// TIA Portal V15.1 export
// export: Created 2024-05-17T05:38:55.7336382Z, ExportSetting WithDefaults, DisplayName Totally Integrated Automation Portal, DisplayVersion V15.1 Update 5, DisplayName TIA Portal Openness, DisplayVersion V15.1 Update 5, DisplayName SINAMICS Startdrive Advanced, DisplayVersion V15.1, DisplayName G130, G150, S120, S150, SINAMICS MV, S210, DisplayVersion V15.1, DisplayName G110M, G120, G120C, G120D, G120P, DisplayVersion V15.1, DisplayName STEP 7 Professional, DisplayVersion V15.1 Update 5, DisplayName STEP 7 Safety, DisplayVersion V15.1, DisplayName WinCC Professional, DisplayVersion V15.1 Update 5, DisplayName SIMATIC Visualization Architect, DisplayVersion V15.1
FUNCTION "209220ZM01Andon" : Void   // FC356, FBD
TITLE = 209220ZM01 Andon
{ S7_Optimized_Access := 'FALSE' }
AUTHOR : VCG
NAME : Mot001
VERSION : 0.1
// stored: AutoNumber false, IsIECCheckEnabled false, SetENOAutomatically False, UDAEnableTagReadback false
   VAR_OUTPUT
      O_AlarmA : Bool;   // Alarm A
      O_AlarmB : Bool;   // Alarm B
      O_AlarmC : Bool;   // Alarm C
      O_AlarmD : Bool;   // Alarm D
      O_AlarmABCondition : Bool;   // Alarms resetable
      H_IAnim : Word;   // Animation bits to Icon in WinCC
   END_VAR
BEGIN

REGION Network 1: **** 1 - Inputs **** HMI Commands
   // HMI Commands from the WinCC
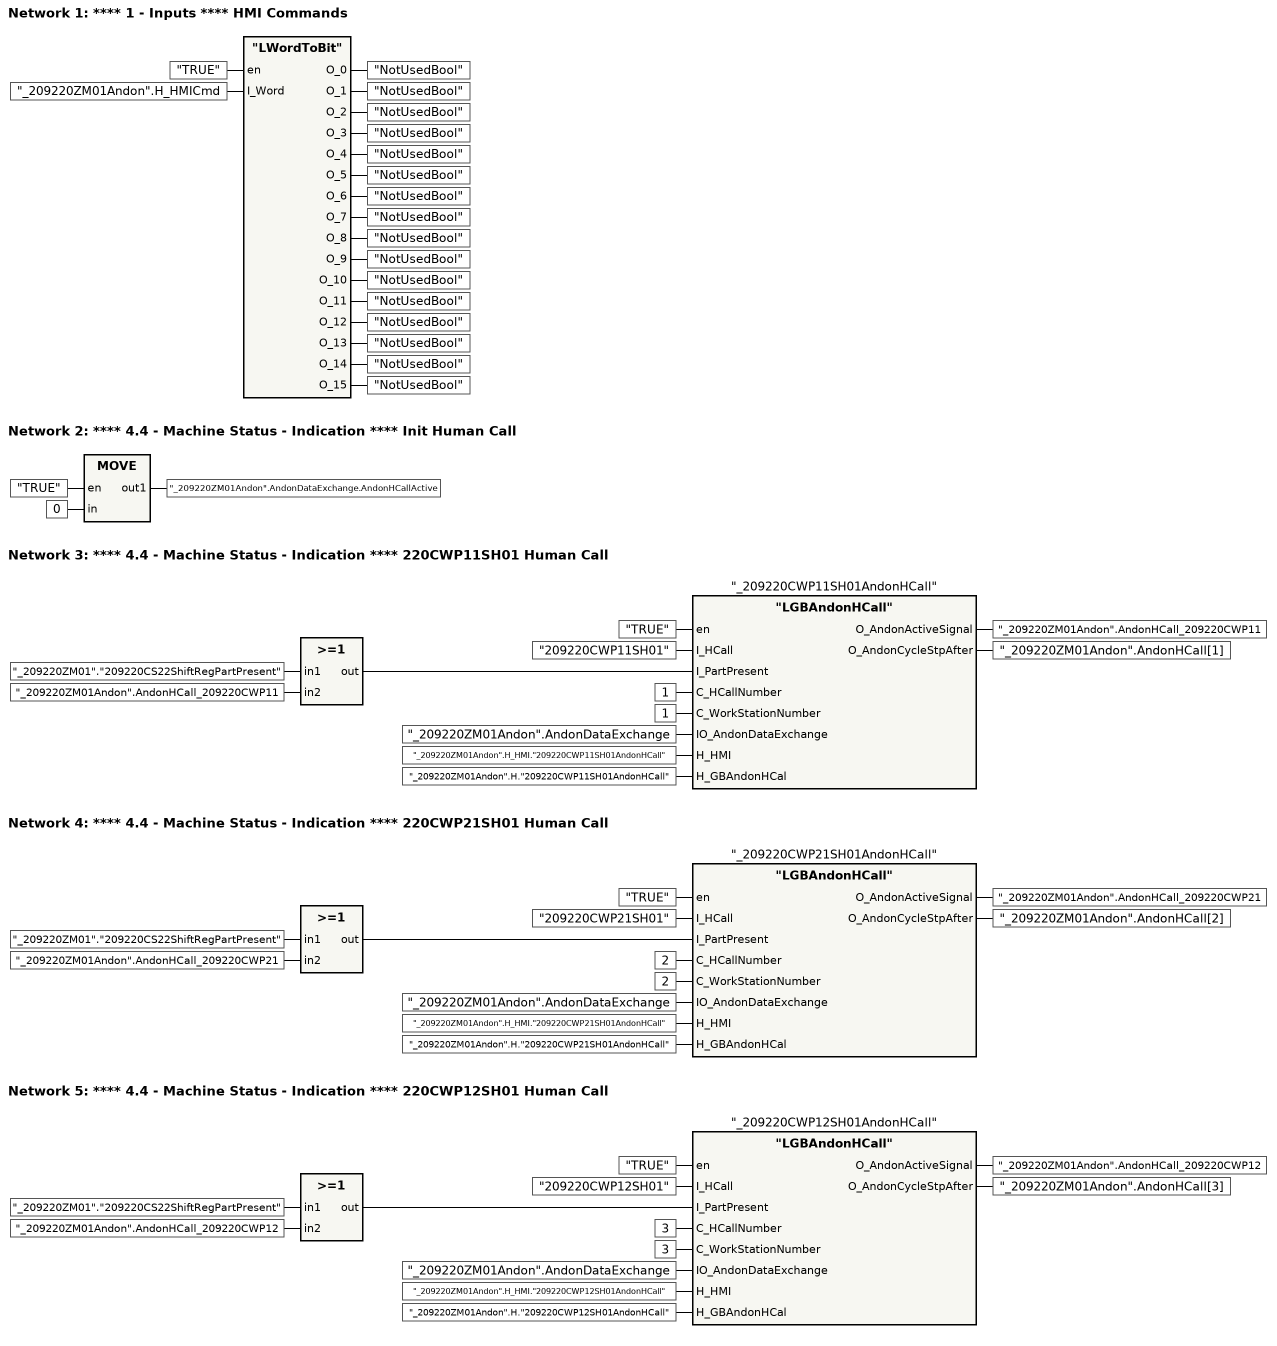
   IF "TRUE" THEN
       "LWordToBit"(I_Word := "_209220ZM01Andon".H_HMICmd,
                    O_0 => "NotUsedBool",
                    O_1 => "NotUsedBool",
                    O_2 => "NotUsedBool",
                    O_3 => "NotUsedBool",
                    O_4 => "NotUsedBool",
                    O_5 => "NotUsedBool",
                    O_6 => "NotUsedBool",
                    O_7 => "NotUsedBool",
                    O_8 => "NotUsedBool",
                    O_9 => "NotUsedBool",
                    O_10 => "NotUsedBool",
                    O_11 => "NotUsedBool",
                    O_12 => "NotUsedBool",
                    O_13 => "NotUsedBool",
                    O_14 => "NotUsedBool",
                    O_15 => "NotUsedBool");
   END_IF;
END_REGION

REGION Network 2: **** 4.4 - Machine Status - Indication **** Init Human Call
   IF "TRUE" THEN "_209220ZM01Andon".AndonDataExchange.AndonHCallActive := 0; END_IF;
END_REGION

REGION Network 3: **** 4.4 - Machine Status - Indication **** 220CWP11SH01 Human Call
   IF "TRUE" THEN
       "_209220CWP11SH01AndonHCall"(I_HCall := "209220CWP11SH01",   // "LGBAndonHCall"
                               I_PartPresent := "_209220ZM01"."209220CS22ShiftRegPartPresent" OR "_209220ZM01Andon".AndonHCall_209220CWP11,
                               C_HCallNumber := 1,
                               C_WorkStationNumber := 1,
                               IO_AndonDataExchange := "_209220ZM01Andon".AndonDataExchange,
                               H_HMI := "_209220ZM01Andon".H_HMI."209220CWP11SH01AndonHCall",
                               H_GBAndonHCal := "_209220ZM01Andon".H."209220CWP11SH01AndonHCall",
                               O_AndonActiveSignal => "_209220ZM01Andon".AndonHCall_209220CWP11,
                               O_AndonCycleStpAfter => "_209220ZM01Andon".AndonHCall[1]);
   END_IF;
END_REGION

REGION Network 4: **** 4.4 - Machine Status - Indication **** 220CWP21SH01 Human Call
   IF "TRUE" THEN
       "_209220CWP21SH01AndonHCall"(I_HCall := "209220CWP21SH01",   // "LGBAndonHCall"
                               I_PartPresent := "_209220ZM01"."209220CS22ShiftRegPartPresent" OR "_209220ZM01Andon".AndonHCall_209220CWP21,
                               C_HCallNumber := 2,
                               C_WorkStationNumber := 2,
                               IO_AndonDataExchange := "_209220ZM01Andon".AndonDataExchange,
                               H_HMI := "_209220ZM01Andon".H_HMI."209220CWP21SH01AndonHCall",
                               H_GBAndonHCal := "_209220ZM01Andon".H."209220CWP21SH01AndonHCall",
                               O_AndonActiveSignal => "_209220ZM01Andon".AndonHCall_209220CWP21,
                               O_AndonCycleStpAfter => "_209220ZM01Andon".AndonHCall[2]);
   END_IF;
END_REGION

REGION Network 5: **** 4.4 - Machine Status - Indication **** 220CWP12SH01 Human Call
   IF "TRUE" THEN
       "_209220CWP12SH01AndonHCall"(I_HCall := "209220CWP12SH01",   // "LGBAndonHCall"
                               I_PartPresent := "_209220ZM01"."209220CS22ShiftRegPartPresent" OR "_209220ZM01Andon".AndonHCall_209220CWP12,
                               C_HCallNumber := 3,
                               C_WorkStationNumber := 3,
                               IO_AndonDataExchange := "_209220ZM01Andon".AndonDataExchange,
                               H_HMI := "_209220ZM01Andon".H_HMI."209220CWP12SH01AndonHCall",
                               H_GBAndonHCal := "_209220ZM01Andon".H."209220CWP12SH01AndonHCall",
                               O_AndonActiveSignal => "_209220ZM01Andon".AndonHCall_209220CWP12,
                               O_AndonCycleStpAfter => "_209220ZM01Andon".AndonHCall[3]);
   END_IF;
END_REGION

REGION Network 6: **** 4.4 - Machine Status - Indication **** 220CWP22SH01 Human Call
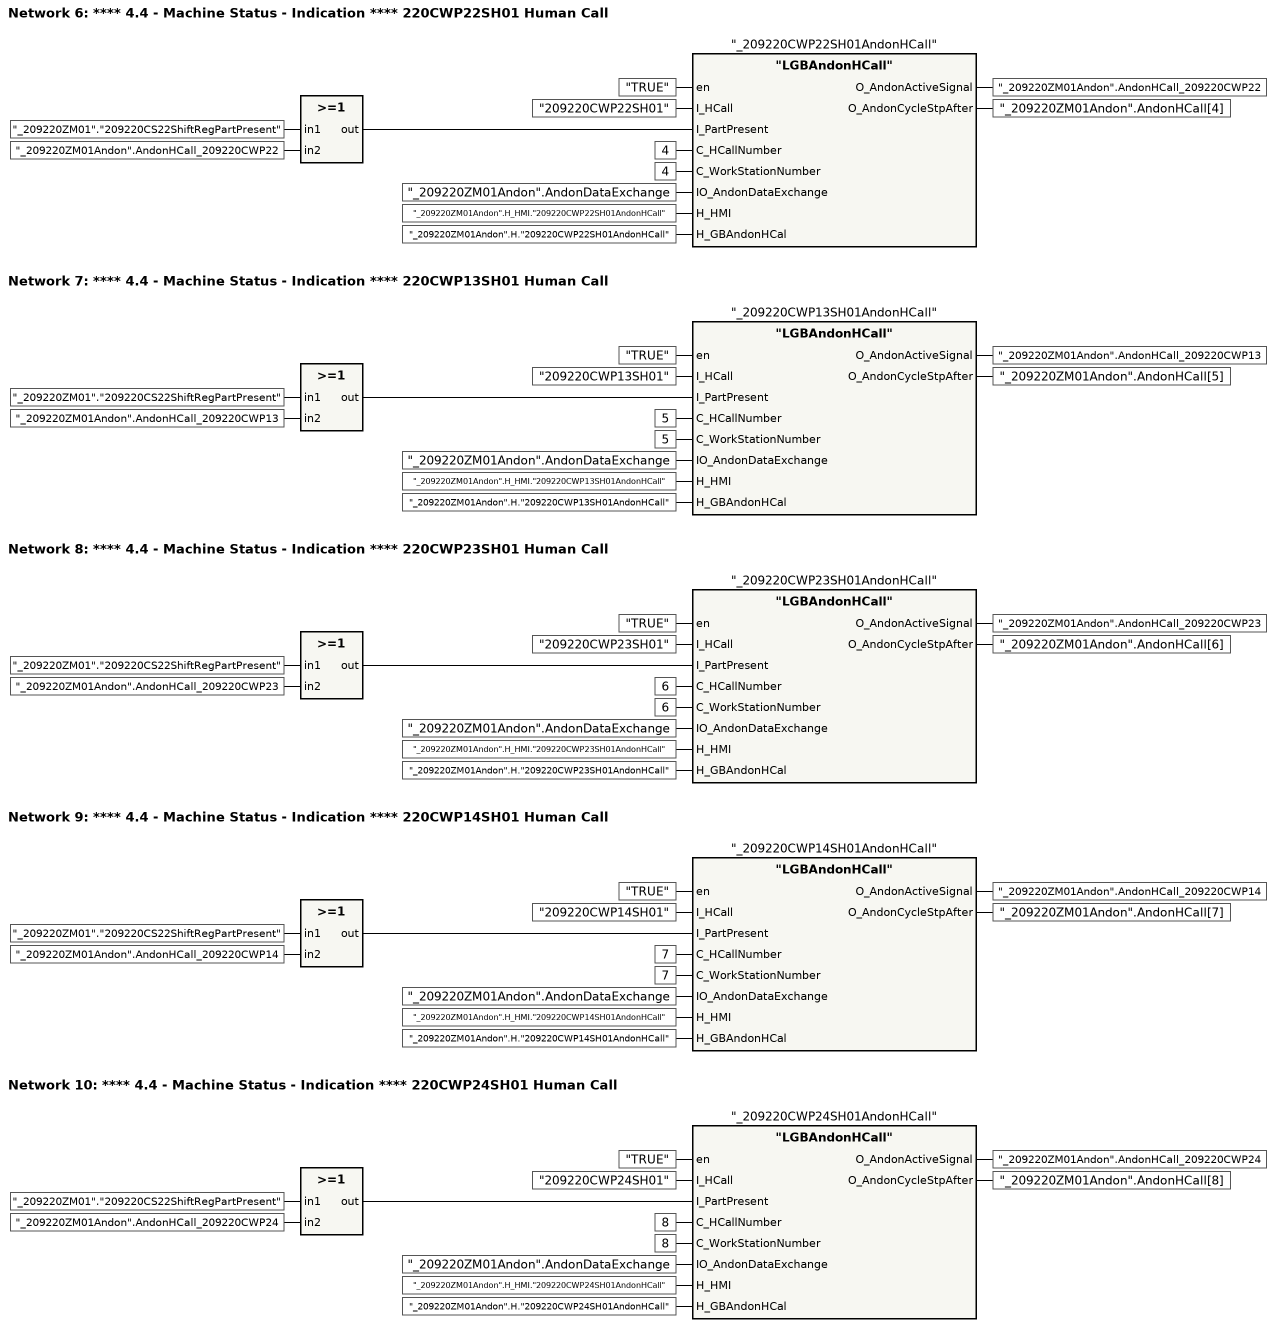
   IF "TRUE" THEN
       "_209220CWP22SH01AndonHCall"(I_HCall := "209220CWP22SH01",   // "LGBAndonHCall"
                               I_PartPresent := "_209220ZM01"."209220CS22ShiftRegPartPresent" OR "_209220ZM01Andon".AndonHCall_209220CWP22,
                               C_HCallNumber := 4,
                               C_WorkStationNumber := 4,
                               IO_AndonDataExchange := "_209220ZM01Andon".AndonDataExchange,
                               H_HMI := "_209220ZM01Andon".H_HMI."209220CWP22SH01AndonHCall",
                               H_GBAndonHCal := "_209220ZM01Andon".H."209220CWP22SH01AndonHCall",
                               O_AndonActiveSignal => "_209220ZM01Andon".AndonHCall_209220CWP22,
                               O_AndonCycleStpAfter => "_209220ZM01Andon".AndonHCall[4]);
   END_IF;
END_REGION

REGION Network 7: **** 4.4 - Machine Status - Indication **** 220CWP13SH01 Human Call
   IF "TRUE" THEN
       "_209220CWP13SH01AndonHCall"(I_HCall := "209220CWP13SH01",   // "LGBAndonHCall"
                               I_PartPresent := "_209220ZM01"."209220CS22ShiftRegPartPresent" OR "_209220ZM01Andon".AndonHCall_209220CWP13,
                               C_HCallNumber := 5,
                               C_WorkStationNumber := 5,
                               IO_AndonDataExchange := "_209220ZM01Andon".AndonDataExchange,
                               H_HMI := "_209220ZM01Andon".H_HMI."209220CWP13SH01AndonHCall",
                               H_GBAndonHCal := "_209220ZM01Andon".H."209220CWP13SH01AndonHCall",
                               O_AndonActiveSignal => "_209220ZM01Andon".AndonHCall_209220CWP13,
                               O_AndonCycleStpAfter => "_209220ZM01Andon".AndonHCall[5]);
   END_IF;
END_REGION

REGION Network 8: **** 4.4 - Machine Status - Indication **** 220CWP23SH01 Human Call
   IF "TRUE" THEN
       "_209220CWP23SH01AndonHCall"(I_HCall := "209220CWP23SH01",   // "LGBAndonHCall"
                               I_PartPresent := "_209220ZM01"."209220CS22ShiftRegPartPresent" OR "_209220ZM01Andon".AndonHCall_209220CWP23,
                               C_HCallNumber := 6,
                               C_WorkStationNumber := 6,
                               IO_AndonDataExchange := "_209220ZM01Andon".AndonDataExchange,
                               H_HMI := "_209220ZM01Andon".H_HMI."209220CWP23SH01AndonHCall",
                               H_GBAndonHCal := "_209220ZM01Andon".H."209220CWP23SH01AndonHCall",
                               O_AndonActiveSignal => "_209220ZM01Andon".AndonHCall_209220CWP23,
                               O_AndonCycleStpAfter => "_209220ZM01Andon".AndonHCall[6]);
   END_IF;
END_REGION

REGION Network 9: **** 4.4 - Machine Status - Indication **** 220CWP14SH01 Human Call
   IF "TRUE" THEN
       "_209220CWP14SH01AndonHCall"(I_HCall := "209220CWP14SH01",   // "LGBAndonHCall"
                               I_PartPresent := "_209220ZM01"."209220CS22ShiftRegPartPresent" OR "_209220ZM01Andon".AndonHCall_209220CWP14,
                               C_HCallNumber := 7,
                               C_WorkStationNumber := 7,
                               IO_AndonDataExchange := "_209220ZM01Andon".AndonDataExchange,
                               H_HMI := "_209220ZM01Andon".H_HMI."209220CWP14SH01AndonHCall",
                               H_GBAndonHCal := "_209220ZM01Andon".H."209220CWP14SH01AndonHCall",
                               O_AndonActiveSignal => "_209220ZM01Andon".AndonHCall_209220CWP14,
                               O_AndonCycleStpAfter => "_209220ZM01Andon".AndonHCall[7]);
   END_IF;
END_REGION

REGION Network 10: **** 4.4 - Machine Status - Indication **** 220CWP24SH01 Human Call
   IF "TRUE" THEN
       "_209220CWP24SH01AndonHCall"(I_HCall := "209220CWP24SH01",   // "LGBAndonHCall"
                               I_PartPresent := "_209220ZM01"."209220CS22ShiftRegPartPresent" OR "_209220ZM01Andon".AndonHCall_209220CWP24,
                               C_HCallNumber := 8,
                               C_WorkStationNumber := 8,
                               IO_AndonDataExchange := "_209220ZM01Andon".AndonDataExchange,
                               H_HMI := "_209220ZM01Andon".H_HMI."209220CWP24SH01AndonHCall",
                               H_GBAndonHCal := "_209220ZM01Andon".H."209220CWP24SH01AndonHCall",
                               O_AndonActiveSignal => "_209220ZM01Andon".AndonHCall_209220CWP24,
                               O_AndonCycleStpAfter => "_209220ZM01Andon".AndonHCall[8]);
   END_IF;
END_REGION

REGION Network 11: **** 4.4 - Machine Status - Indication **** 220CWP15SH01 Human Call
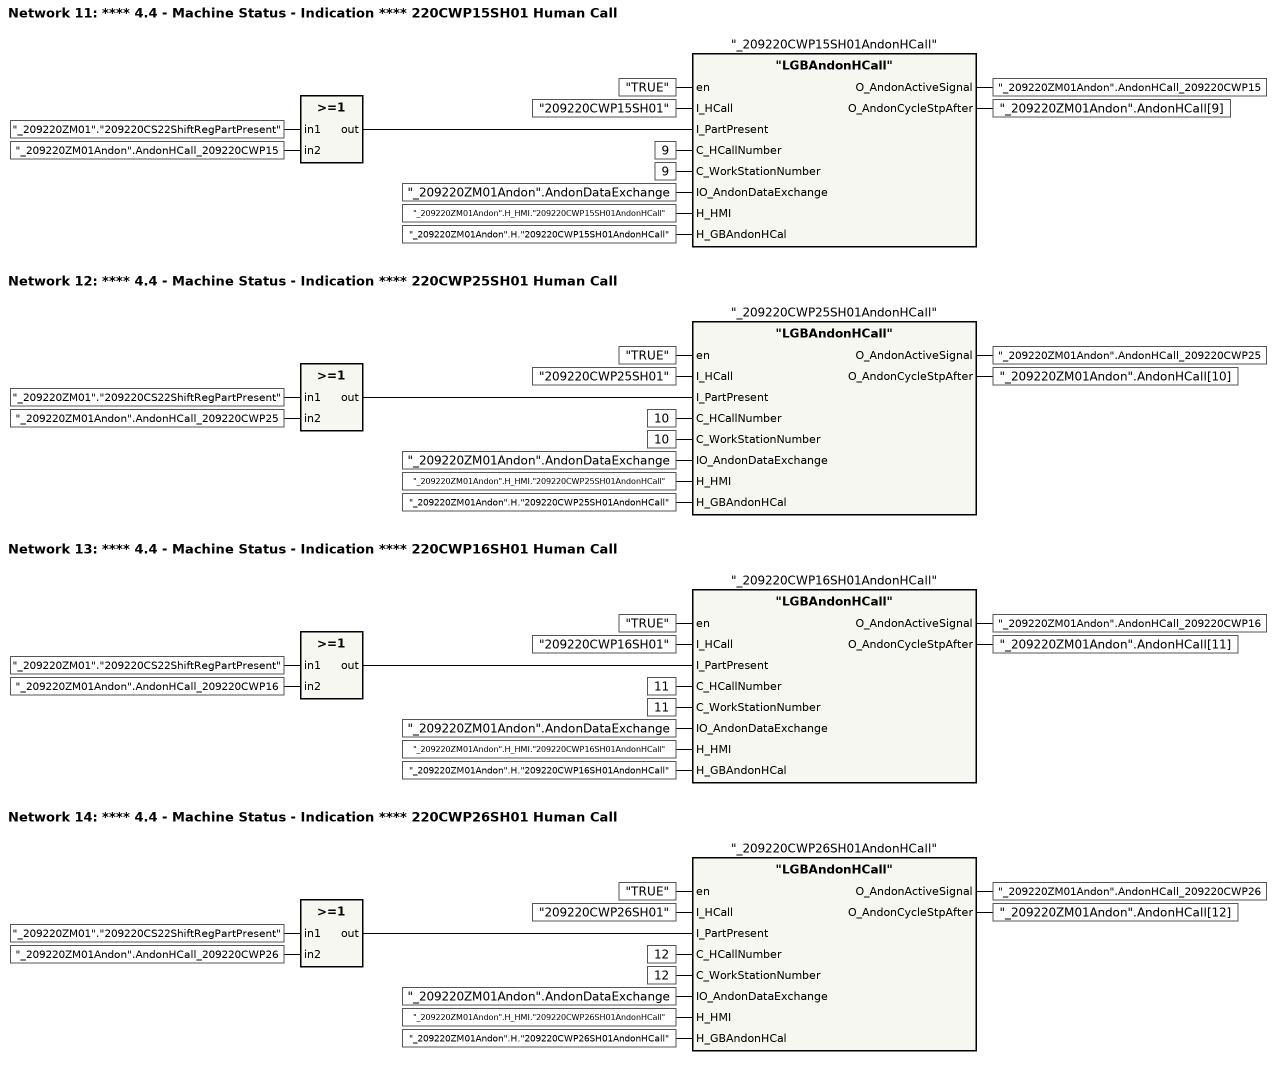
   IF "TRUE" THEN
       "_209220CWP15SH01AndonHCall"(I_HCall := "209220CWP15SH01",   // "LGBAndonHCall"
                               I_PartPresent := "_209220ZM01"."209220CS22ShiftRegPartPresent" OR "_209220ZM01Andon".AndonHCall_209220CWP15,
                               C_HCallNumber := 9,
                               C_WorkStationNumber := 9,
                               IO_AndonDataExchange := "_209220ZM01Andon".AndonDataExchange,
                               H_HMI := "_209220ZM01Andon".H_HMI."209220CWP15SH01AndonHCall",
                               H_GBAndonHCal := "_209220ZM01Andon".H."209220CWP15SH01AndonHCall",
                               O_AndonActiveSignal => "_209220ZM01Andon".AndonHCall_209220CWP15,
                               O_AndonCycleStpAfter => "_209220ZM01Andon".AndonHCall[9]);
   END_IF;
END_REGION

REGION Network 12: **** 4.4 - Machine Status - Indication **** 220CWP25SH01 Human Call
   IF "TRUE" THEN
       "_209220CWP25SH01AndonHCall"(I_HCall := "209220CWP25SH01",   // "LGBAndonHCall"
                               I_PartPresent := "_209220ZM01"."209220CS22ShiftRegPartPresent" OR "_209220ZM01Andon".AndonHCall_209220CWP25,
                               C_HCallNumber := 10,
                               C_WorkStationNumber := 10,
                               IO_AndonDataExchange := "_209220ZM01Andon".AndonDataExchange,
                               H_HMI := "_209220ZM01Andon".H_HMI."209220CWP25SH01AndonHCall",
                               H_GBAndonHCal := "_209220ZM01Andon".H."209220CWP25SH01AndonHCall",
                               O_AndonActiveSignal => "_209220ZM01Andon".AndonHCall_209220CWP25,
                               O_AndonCycleStpAfter => "_209220ZM01Andon".AndonHCall[10]);
   END_IF;
END_REGION

REGION Network 13: **** 4.4 - Machine Status - Indication **** 220CWP16SH01 Human Call
   IF "TRUE" THEN
       "_209220CWP16SH01AndonHCall"(I_HCall := "209220CWP16SH01",   // "LGBAndonHCall"
                               I_PartPresent := "_209220ZM01"."209220CS22ShiftRegPartPresent" OR "_209220ZM01Andon".AndonHCall_209220CWP16,
                               C_HCallNumber := 11,
                               C_WorkStationNumber := 11,
                               IO_AndonDataExchange := "_209220ZM01Andon".AndonDataExchange,
                               H_HMI := "_209220ZM01Andon".H_HMI."209220CWP16SH01AndonHCall",
                               H_GBAndonHCal := "_209220ZM01Andon".H."209220CWP16SH01AndonHCall",
                               O_AndonActiveSignal => "_209220ZM01Andon".AndonHCall_209220CWP16,
                               O_AndonCycleStpAfter => "_209220ZM01Andon".AndonHCall[11]);
   END_IF;
END_REGION

REGION Network 14: **** 4.4 - Machine Status - Indication **** 220CWP26SH01 Human Call
   IF "TRUE" THEN
       "_209220CWP26SH01AndonHCall"(I_HCall := "209220CWP26SH01",   // "LGBAndonHCall"
                               I_PartPresent := "_209220ZM01"."209220CS22ShiftRegPartPresent" OR "_209220ZM01Andon".AndonHCall_209220CWP26,
                               C_HCallNumber := 12,
                               C_WorkStationNumber := 12,
                               IO_AndonDataExchange := "_209220ZM01Andon".AndonDataExchange,
                               H_HMI := "_209220ZM01Andon".H_HMI."209220CWP26SH01AndonHCall",
                               H_GBAndonHCal := "_209220ZM01Andon".H."209220CWP26SH01AndonHCall",
                               O_AndonActiveSignal => "_209220ZM01Andon".AndonHCall_209220CWP26,
                               O_AndonCycleStpAfter => "_209220ZM01Andon".AndonHCall[12]);
   END_IF;
END_REGION

REGION Network 15: **** 4.4 - Machine Status - Calculation **** Stop Request by Andon HCall
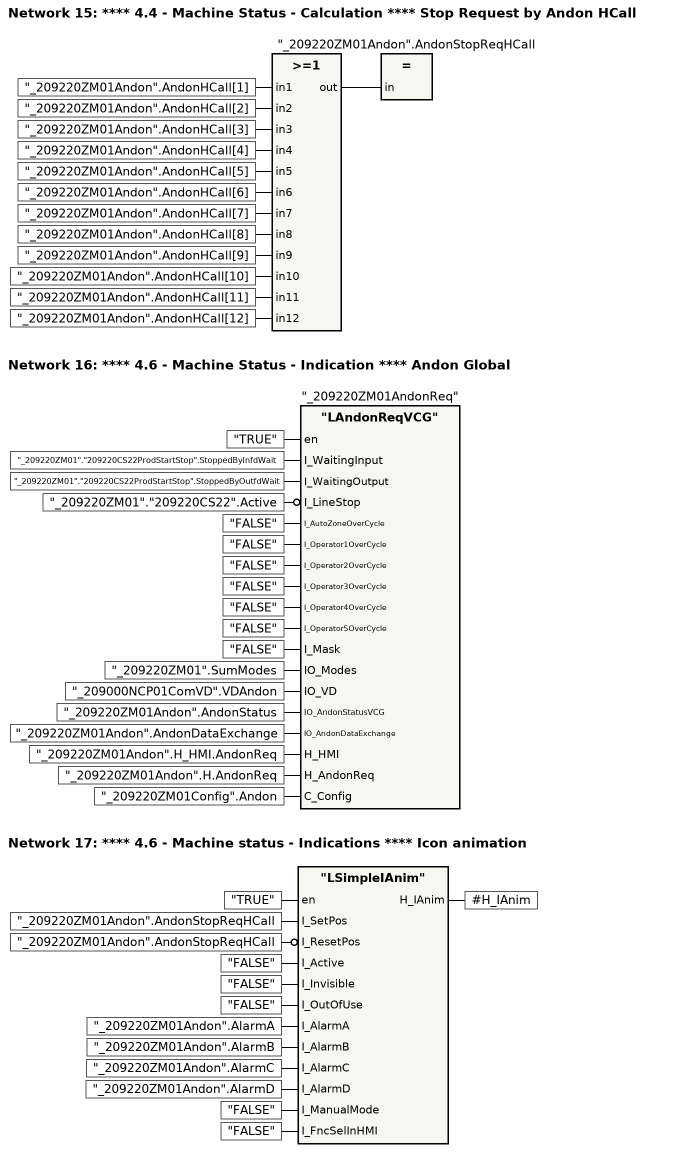
   "_209220ZM01Andon".AndonStopReqHCall := "_209220ZM01Andon".AndonHCall[1] OR "_209220ZM01Andon".AndonHCall[2] OR "_209220ZM01Andon".AndonHCall[3] OR "_209220ZM01Andon".AndonHCall[4] OR "_209220ZM01Andon".AndonHCall[5] OR "_209220ZM01Andon".AndonHCall[6] OR "_209220ZM01Andon".AndonHCall[7] OR "_209220ZM01Andon".AndonHCall[8] OR "_209220ZM01Andon".AndonHCall[9] OR "_209220ZM01Andon".AndonHCall[10] OR "_209220ZM01Andon".AndonHCall[11] OR "_209220ZM01Andon".AndonHCall[12];
END_REGION

REGION Network 16: **** 4.6 - Machine Status - Indication **** Andon Global
   // Request Andon Call
   IF "TRUE" THEN
       "_209220ZM01AndonReq"(I_WaitingInput := "_209220ZM01"."209220CS22ProdStartStop".StoppedByInfdWait,   // "LAndonReqVCG"
                             I_WaitingOutput := "_209220ZM01"."209220CS22ProdStartStop".StoppedByOutfdWait,
                             I_LineStop := NOT "_209220ZM01"."209220CS22".Active,
                             I_AutoZoneOverCycle := "FALSE",
                             I_Operator1OverCycle := "FALSE",
                             I_Operator2OverCycle := "FALSE",
                             I_Operator3OverCycle := "FALSE",
                             I_Operator4OverCycle := "FALSE",
                             I_Operator5OverCycle := "FALSE",
                             I_Mask := "FALSE",
                             IO_Modes := "_209220ZM01".SumModes,
                             IO_VD := "_209000NCP01ComVD".VDAndon,
                             IO_AndonStatusVCG := "_209220ZM01Andon".AndonStatus,
                             IO_AndonDataExchange := "_209220ZM01Andon".AndonDataExchange,
                             H_HMI := "_209220ZM01Andon".H_HMI.AndonReq,
                             H_AndonReq := "_209220ZM01Andon".H.AndonReq,
                             C_Config := "_209220ZM01Config".Andon);
   END_IF;
END_REGION

REGION Network 17: **** 4.6 - Machine status - Indications **** Icon animation
   // Icon animation
   IF "TRUE" THEN
       "LSimpleIAnim"(I_SetPos := "_209220ZM01Andon".AndonStopReqHCall,
                      I_ResetPos := NOT "_209220ZM01Andon".AndonStopReqHCall,
                      I_Active := "FALSE",
                      I_Invisible := "FALSE",
                      I_OutOfUse := "FALSE",
                      I_AlarmA := "_209220ZM01Andon".AlarmA,
                      I_AlarmB := "_209220ZM01Andon".AlarmB,
                      I_AlarmC := "_209220ZM01Andon".AlarmC,
                      I_AlarmD := "_209220ZM01Andon".AlarmD,
                      I_ManualMode := "FALSE",
                      I_FncSelInHMI := "FALSE",
                      H_IAnim => #H_IAnim);
   END_IF;
END_REGION

REGION Network 18: **** 4.6 - Machine status - Indications **** Animation
   // Animation
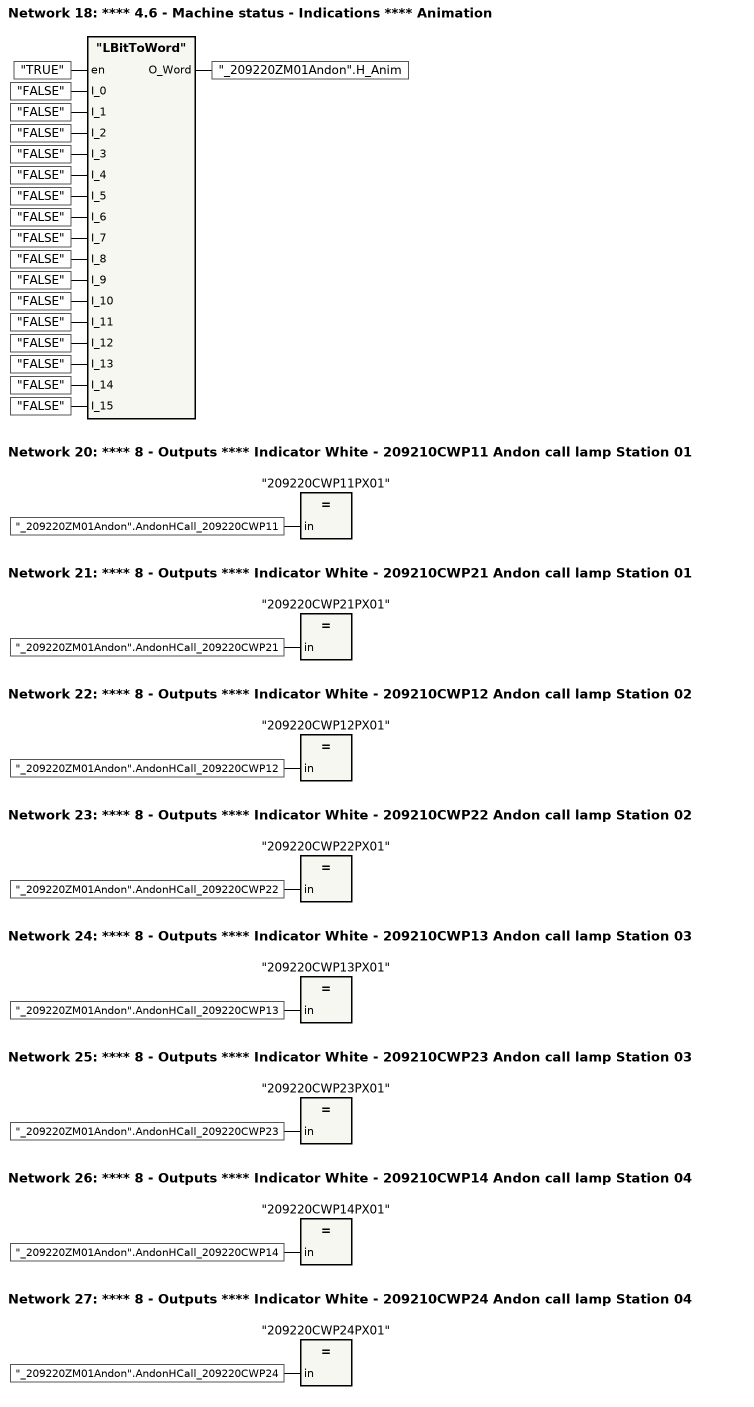
   IF "TRUE" THEN
       "LBitToWord"(I_0 := "FALSE",
                    I_1 := "FALSE",
                    I_2 := "FALSE",
                    I_3 := "FALSE",
                    I_4 := "FALSE",
                    I_5 := "FALSE",
                    I_6 := "FALSE",
                    I_7 := "FALSE",
                    I_8 := "FALSE",
                    I_9 := "FALSE",
                    I_10 := "FALSE",
                    I_11 := "FALSE",
                    I_12 := "FALSE",
                    I_13 := "FALSE",
                    I_14 := "FALSE",
                    I_15 := "FALSE",
                    O_Word => "_209220ZM01Andon".H_Anim);
   END_IF;
END_REGION

NETWORK
TITLE = **** 4.6 - Machine Status - Indications **** Animation DB number
// DB number
      OPN   "_209220ZM01Andon";
      L     DBNO;
      T     "_209220ZM01Andon".H_DBnr;

REGION Network 20: **** 8 - Outputs **** Indicator White - 209210CWP11 Andon call lamp Station 01
   "209220CWP11PX01" := "_209220ZM01Andon".AndonHCall_209220CWP11;
END_REGION

REGION Network 21: **** 8 - Outputs **** Indicator White - 209210CWP21 Andon call lamp Station 01
   "209220CWP21PX01" := "_209220ZM01Andon".AndonHCall_209220CWP21;
END_REGION

REGION Network 22: **** 8 - Outputs **** Indicator White - 209210CWP12 Andon call lamp Station 02
   "209220CWP12PX01" := "_209220ZM01Andon".AndonHCall_209220CWP12;
END_REGION

REGION Network 23: **** 8 - Outputs **** Indicator White - 209210CWP22 Andon call lamp Station 02
   "209220CWP22PX01" := "_209220ZM01Andon".AndonHCall_209220CWP22;
END_REGION

REGION Network 24: **** 8 - Outputs **** Indicator White - 209210CWP13 Andon call lamp Station 03
   "209220CWP13PX01" := "_209220ZM01Andon".AndonHCall_209220CWP13;
END_REGION

REGION Network 25: **** 8 - Outputs **** Indicator White - 209210CWP23 Andon call lamp Station 03
   "209220CWP23PX01" := "_209220ZM01Andon".AndonHCall_209220CWP23;
END_REGION

REGION Network 26: **** 8 - Outputs **** Indicator White - 209210CWP14 Andon call lamp Station 04
   "209220CWP14PX01" := "_209220ZM01Andon".AndonHCall_209220CWP14;
END_REGION

REGION Network 27: **** 8 - Outputs **** Indicator White - 209210CWP24 Andon call lamp Station 04
   "209220CWP24PX01" := "_209220ZM01Andon".AndonHCall_209220CWP24;
END_REGION

REGION Network 28: **** 8 - Outputs **** Indicator White - 209210CWP15 Andon call lamp Station 05
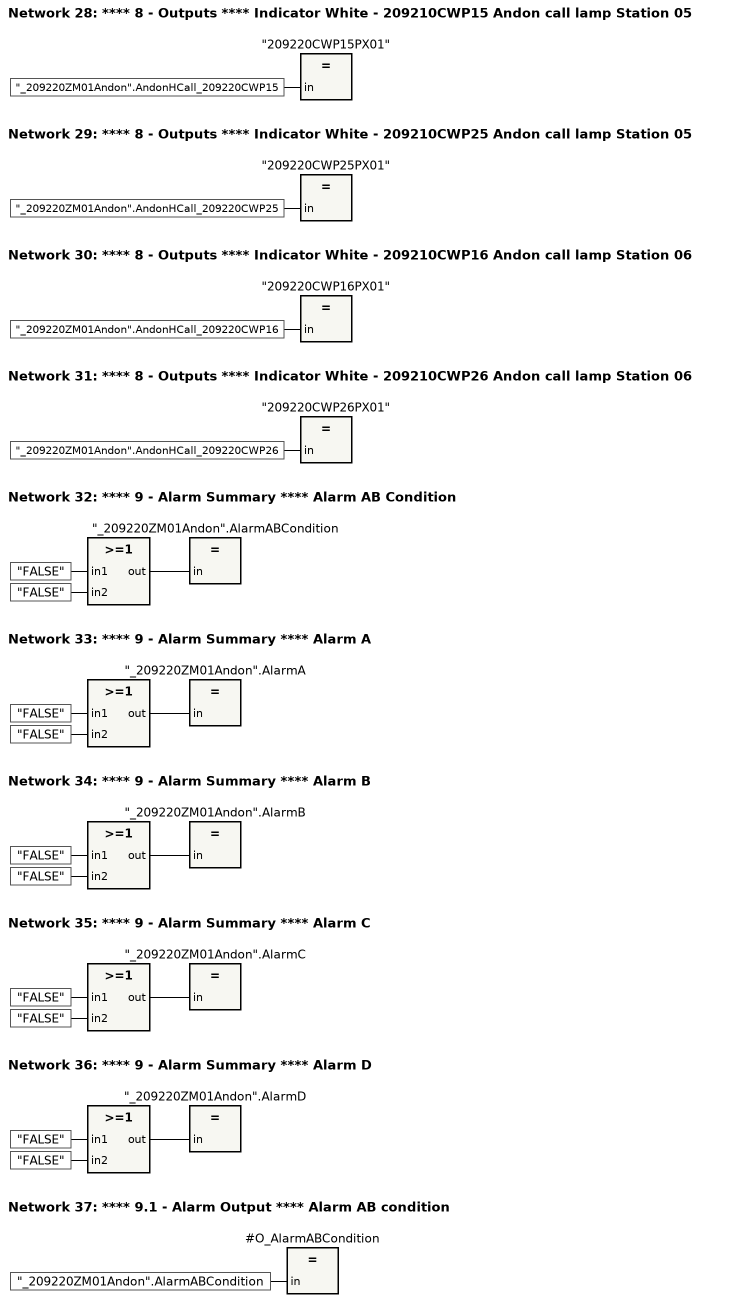
   "209220CWP15PX01" := "_209220ZM01Andon".AndonHCall_209220CWP15;
END_REGION

REGION Network 29: **** 8 - Outputs **** Indicator White - 209210CWP25 Andon call lamp Station 05
   "209220CWP25PX01" := "_209220ZM01Andon".AndonHCall_209220CWP25;
END_REGION

REGION Network 30: **** 8 - Outputs **** Indicator White - 209210CWP16 Andon call lamp Station 06
   "209220CWP16PX01" := "_209220ZM01Andon".AndonHCall_209220CWP16;
END_REGION

REGION Network 31: **** 8 - Outputs **** Indicator White - 209210CWP26 Andon call lamp Station 06
   "209220CWP26PX01" := "_209220ZM01Andon".AndonHCall_209220CWP26;
END_REGION

REGION Network 32: **** 9 - Alarm Summary **** Alarm AB Condition
   // Alarm AB condition
   "_209220ZM01Andon".AlarmABCondition := "FALSE" OR "FALSE";
END_REGION

REGION Network 33: **** 9 - Alarm Summary **** Alarm A
   // Summary of alarms A
   "_209220ZM01Andon".AlarmA := "FALSE" OR "FALSE";
END_REGION

REGION Network 34: **** 9 - Alarm Summary **** Alarm B
   // Summary of alarms B
   "_209220ZM01Andon".AlarmB := "FALSE" OR "FALSE";
END_REGION

REGION Network 35: **** 9 - Alarm Summary **** Alarm C
   // Summary of alarms C
   "_209220ZM01Andon".AlarmC := "FALSE" OR "FALSE";
END_REGION

REGION Network 36: **** 9 - Alarm Summary **** Alarm D
   // Summary of alarms D
   "_209220ZM01Andon".AlarmD := "FALSE" OR "FALSE";
END_REGION

REGION Network 37: **** 9.1 - Alarm Output **** Alarm AB condition
   // Alarm AB condition
   #O_AlarmABCondition := "_209220ZM01Andon".AlarmABCondition;
END_REGION

REGION Network 38: **** 9.1 - Alarm Output **** Alarm A
   // Output Alarm A
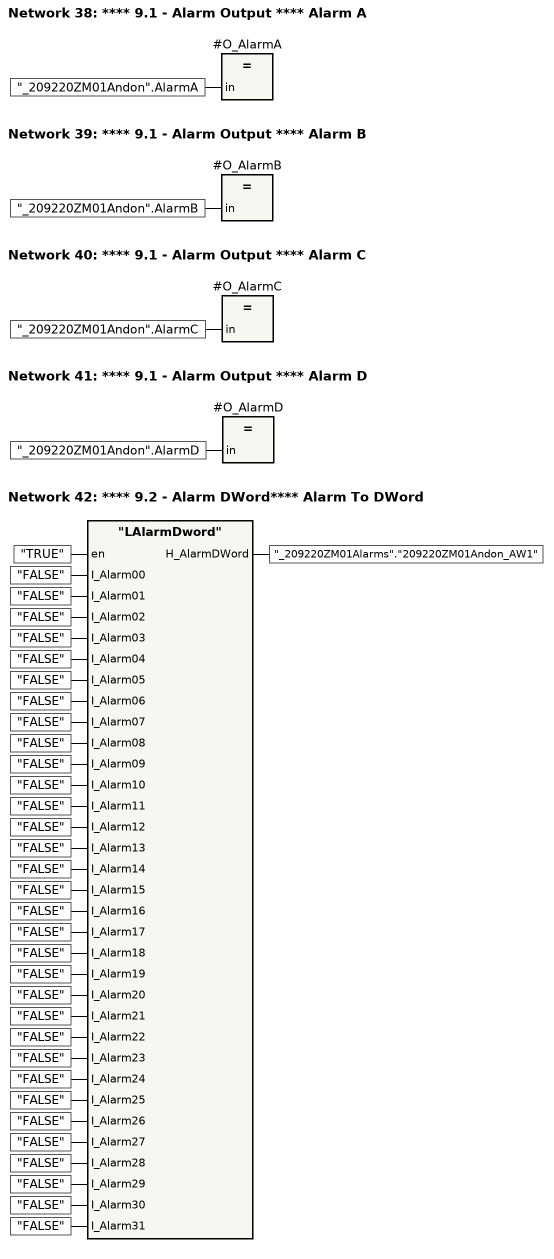
   #O_AlarmA := "_209220ZM01Andon".AlarmA;
END_REGION

REGION Network 39: **** 9.1 - Alarm Output **** Alarm B
   // Output Alarm B
   #O_AlarmB := "_209220ZM01Andon".AlarmB;
END_REGION

REGION Network 40: **** 9.1 - Alarm Output **** Alarm C
   // Output Alarm A
   #O_AlarmC := "_209220ZM01Andon".AlarmC;
END_REGION

REGION Network 41: **** 9.1 - Alarm Output **** Alarm D
   // Output Alarm D
   #O_AlarmD := "_209220ZM01Andon".AlarmD;
END_REGION

REGION Network 42: **** 9.2 - Alarm DWord**** Alarm To DWord
   // Alarm Word
   IF "TRUE" THEN
       "LAlarmDword"(I_Alarm00 := "FALSE",
                     I_Alarm01 := "FALSE",
                     I_Alarm02 := "FALSE",
                     I_Alarm03 := "FALSE",
                     I_Alarm04 := "FALSE",
                     I_Alarm05 := "FALSE",
                     I_Alarm06 := "FALSE",
                     I_Alarm07 := "FALSE",
                     I_Alarm08 := "FALSE",
                     I_Alarm09 := "FALSE",
                     I_Alarm10 := "FALSE",
                     I_Alarm11 := "FALSE",
                     I_Alarm12 := "FALSE",
                     I_Alarm13 := "FALSE",
                     I_Alarm14 := "FALSE",
                     I_Alarm15 := "FALSE",
                     I_Alarm16 := "FALSE",
                     I_Alarm17 := "FALSE",
                     I_Alarm18 := "FALSE",
                     I_Alarm19 := "FALSE",
                     I_Alarm20 := "FALSE",
                     I_Alarm21 := "FALSE",
                     I_Alarm22 := "FALSE",
                     I_Alarm23 := "FALSE",
                     I_Alarm24 := "FALSE",
                     I_Alarm25 := "FALSE",
                     I_Alarm26 := "FALSE",
                     I_Alarm27 := "FALSE",
                     I_Alarm28 := "FALSE",
                     I_Alarm29 := "FALSE",
                     I_Alarm30 := "FALSE",
                     I_Alarm31 := "FALSE",
                     H_AlarmDWord => "_209220ZM01Alarms"."209220ZM01Andon_AW1");
   END_IF;
END_REGION
END_FUNCTION
